// TIA Portal V19 export
DATA_BLOCK "PitTable1"   // DB187
// stored: InstanceOfName PitTable1_FB, InstanceOfType FB
"PitTable1_FB"
   // VAR_INPUT
   //    AreaInterface : "AreaInterface";
   //    ZSI : "udt_ZoneSafetyInterface";
   //    DSI : "udt_DeviceSafetyInterface";
   //    DataIn : Struct
   //       Pb_Up : Bool;
   //       Pb_Dwn : Bool;
   //       Ls_Up : Bool;
   //       Ls_Down : Bool;
   //    END_STRUCT;
   //    CIn : Struct
   //       Manager : "ValveMachine_Manager";
   //       ExtEnable_Up : Bool;
   //       ExtEnable_Down : Bool;
   //    END_STRUCT;
   //    Config : Struct
   //       LIFT : "ValveMachine_Config";
   //       Exist : Bool;
   //    END_STRUCT;
   // END_VAR
   // VAR_OUTPUT
   //    MachineInterface : "MachineInterface";
   //    DataOut : Struct
   //       V_Up : Bool;
   //       V_Down : Bool;
   //       Lamp : Bool;
   //    END_STRUCT;
   // END_VAR
   // VAR
   //    Warning : "ValveMachine_Wng";
   //    Alarm : "ValveAlr";
   //    Lift : "ValveMachine_FB";
   //    TimerRestManualReq : TON_TIME;
   // END_VAR
BEGIN
END_DATA_BLOCK
